VISUALIZATION HMI  // 2x2
END_VISUALIZATION

(* stored: Version 1.1.0.1, ProductVersion 3.1.4024.12
   Visu HMI: Id {4ba6f969-e9a8-45bf-a479-56a651a372f9} *)
